{attribute 'qualified_only'}
{attribute 'strict'}
TYPE E_WorkingStates ://can't divide into 2 states for load and unload,for sometimes if not unload,then call load,can cause accident
(
	IDLE := 0,
	INIT,
	CHECK,
	WAIT_NEW_TOTE,
	LOADING,
	WAIT_FINISHED,
	TOTE_LOAD,
	TOTE_UNLOAD,
	BAG_OPEN,
	BAG_CLOSE,
	TOTE_LIFT_UP,
	TOTE_LIFT_DOWN,
	BAG_OPEN_UP,
	BAG_OPEN_DOWN,
	TOTE_OUT,
	WAIT_1,
	
	
	BAG_OPEN_HOME,//CYLINDER AND AXIS HOME
	BAG_OPEN_VACUUN_BEGIN,
	VACUUN_ON,
	VACUUN_OFF,
	BAG_OPEN_VACUUN_END,
	BAG_OPEN_SIDE_CYCLINDER_DOWN,
	BAG_OPEN_SIDE_CYCLINDER_UP,
	BAG_OPEN_SIDE_CYCLINDER_EXTEND,
	BAG_OPEN_SIDE_CYCLINDER_RETRACT,
	BAG_OPEN_AXIS_CYCLINDER_DOWN,
	BAG_OPEN_AXIS_CYCLINDER_UP,
	BAG_OPEN_AXIS_CLOSE,
	BAG_OPEN_AXIS_OPEN,
	
	
	AGING_STATE_0,
	AGING_STATE_1,
	
	
	
	
	WAIT,
	
	WAIT_UNLOADING,
	WAIT_SENSOR_ON,
	WAIT_SENSOR_OFF,	
	DONE				:= 100,
	ERROR				:= 200
	
);
END_TYPE

(* stored: Version 1.1.0.1, ProductVersion 3.1.4024.12
   DUT E_WorkingStates: Id {6f75a5c4-44ff-4fb1-9d15-0d913b000b2e} *)
